# EPICS StreamDevice protocol: CavitySimulator-loc/CavitySimulatorApp/Db/Calibration.proto
ExtraInpout = Ignore;
InTerminator = NL;
OutTerminator = NL"*OPC?"NL;

calibrate{ out "CAL:VM\$1";}
